# EPICS autosave request: exampleApp/Db/ADCSimDetectorN_settings.req
$(P)$(R)Amplitude
$(P)$(R)Offset
$(P)$(R)Frequency
$(P)$(R)Phase
$(P)$(R)Noise
